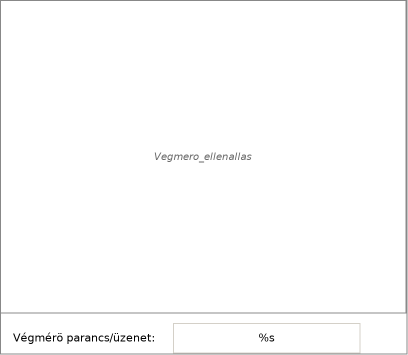
VISUALIZATION Vegmero_auto  // 408x355
    TabControl (0,0 406x313)
        shows Vegmero_ellenallas()
        shows Vegmero_szigeteles()
        shows Vegmero_idoallando()
        shows Vegmero_sokk()
        shows Vegmero_teljes()
        shows Vegmero_etalon()
        [0]: TabTitle=Ellenállás
        [1]: TabTitle=Szigetelés
        [2]: TabTitle=Idöállandó
        [3]: TabTitle=Sokk
        [4]: TabTitle=Teljes/Etalon
        [5]: TabTitle=Etalon
    Textfield (173,323 187x30), "%s", text variable: VEGMERO.s_InCommand
    Label (8,328 150x20), "Végmérö parancs/üzenet:"
END_VISUALIZATION

(* stored: Version 1.1.0.1, ProductVersion 3.1.4024.11
   Visu Vegmero_auto: Id {c69f0959-2fce-4a47-81c2-6b6119b70e72} *)
